INTERFACE I_Signal EXTENDS I_Debug, I_Tagged

METHOD Pair : Result
VAR_INPUT
	iReceiver		: I_Receiver;
END_VAR
END_METHOD

METHOD Unpair : Result
VAR_INPUT
	iReceiver		: I_Receiver;
END_VAR
END_METHOD

END_INTERFACE

(* stored: Version 1.1.0.1
   Itf I_Signal: Id {24f70e98-e98e-42d2-be1a-1b78aa21ba77}
   Method Pair: Id {ca87eecf-5514-49b6-9ee7-6f01e2786d2f}
   Method Unpair: Id {fa23d0f6-12ae-44be-a780-a181f4365fc2} *)
